FUNCTION_BLOCK FB_SlitPair_1
VAR_INPUT
    iBladeNegative: UINT; //Axis ID for negatively positioned blade
    iBladePositive: UINT; //Axis ID for positively positioned blade
    iGapSize: UINT; //Axis ID for the size of gap between slit blades
    iGapCentre: UINT; //Axis ID for the centre position of the gap formed by slit blades
    bEnable: BOOL; //Enable/disable the slit set
    bReset: BOOL; //Reset the slit set
    fEncoderScaling: LREAL := 10000; //default scaling denominator of 10000
    bAutoHome: BOOL := FALSE;
END_VAR
VAR_OUTPUT
    bEnabled: BOOL := FALSE; //Enabled status of function
    bError: BOOL; //Error status of function
    bHoming: BOOL := FALSE; //TRUE if function is homing axes
END_VAR
VAR
    eSlitPairState: E_SlitPairStates := E_SlitPairStates.INIT; //statemachine index

//Internal statuses for logic
    bResetting: BOOL := FALSE; //TRUE if axis going through a reset
    bRealAxesEnabled: BOOL := FALSE; //TRUE if all axes enabled
    bBladesHomed: BOOL:= FALSE; //TRUE if blade axes are calibrated
    bGapHomed: BOOL:= FALSE; //TRUE if virtual axes are calibrated
    bBladesCoupled: BOOL:= FALSE; //TRUE if both blade axes are coupled
    bBladesUncoupled: BOOL := FALSE; //TRUE if both blade axes are uncoupled
    bAxisErrorsPresent: BOOL := FALSE; //TRUE if error present on any real or virtual axis
    bFunctionInErrorState: BOOL := FALSE; //TRUE if function block is in one of the error related states
    fGapSizePosition: LREAL;
    iGapSizePosition AT %Q*: UDINT := 0;
    fGapCentrePosition: LREAL;
    iGapCentrePosition AT %Q*: UDINT := 0;
    resetCounterTimeout: UINT :=0;
    mcHomeGapSize: MC_Home;
    mcHomeGapCentre: MC_Home;
	fbSetPosGapsize: MC_SetPosition;
	fbSetPosGapCentre: MC_SetPosition;
	bSetPosiotnGap: BOOL := FALSE;
END_VAR

(* NOTES
For the virtual axis setup, the encoders need their type changed from "simulation encoder" to "Encoder (Universal)".
In addition the scale factor needs to be changed to a numerator of 1 and denominator of fEncoderScaling which is 10,000 by default)
Care needs to be taken with scaling and setup of both real and virtual axes to ensure velocities are not too fast and axes have time to settle before they submit a "complete move"
*)

//Configure homing routine of virtual axes
GVL.astAxes[iGapSize].stConfig.eHomeSeq := E_HomingRoutines.eHomeDirect;
GVL.astAxes[iGapCentre].stConfig.eHomeSeq := E_HomingRoutines.eHomeDirect;

//Run actions for slit set
actRunMethods(); //Update statuses
actErrorHandling(); //Error handling subroutine
actGapLimits(); //Set virtual axis limits to TRUE
actVirtualAxisPositions(); //Virtual axis encoder position subroutine


//Mc_Home FBs configured to clear homing signal
mcHomeGapSize(Axis := astAxes[iGapSize].Axis, HomingMode:=MC_HomingMode.MC_ResetCalibration);
mcHomeGapCentre(Axis:=astAxes[iGapCentre].Axis, HomingMode:=MC_HomingMode.MC_ResetCalibration);
mcHomeGapSize.Execute := FALSE;
mcHomeGapCentre.Execute := FALSE;

CASE eSlitPairState OF
    E_SlitPairStates.INIT:
        IF bEnable THEN
            eSlitPairState := E_SlitPairStates.INIT_CLEAR_GEARING;
        END_IF

    E_SlitPairStates.INIT_CLEAR_GEARING:
        actClearSlitGearing();
        eSlitPairState := E_SlitPairStates.INIT_GEAROUT_CHECK;

    E_SlitPairStates.INIT_GEAROUT_CHECK: //Check gearOut completion
        IF bBladesUncoupled THEN
            eSlitPairState := E_SlitPairStates.CHECK_HOME_STATUS;
        END_IF

    E_SlitPairStates.CHECK_HOME_STATUS: //If blades are already homed, skip to virtual homing, if blades not homed and autohome enabled then home blades, otherwise wait for blades to be homed
        IF bBladesHomed THEN
			eSlitPairState := E_SlitPairStates.HOME_GAP;
        ELSIF bRealAxesEnabled AND bAutoHome THEN
            eSlitPairState := E_SlitPairStates.HOME_BLADES; //If autohome enabled, home the blades
        END_IF

    E_SlitPairStates.HOME_BLADES: //Initiate homing of blade axes. Homing routine must be pre-configured by user
		mcHomeGapSize.Execute := TRUE;
        mcHomeGapCentre.Execute := TRUE;
        IF mcHomeGapSize.Done AND mcHomeGapCentre.Done THEN
       		GVL.astAxes[iBladeNegative].stControl.eCommand := E_MotionFunctions.eHome;
        	GVL.astAxes[iBladePositive].stControl.eCommand := E_MotionFunctions.eHome;
        	GVL.astAxes[iBladeNegative].stControl.bExecute := TRUE;
        	GVL.astAxes[iBladePositive].stControl.bExecute := TRUE;
        	bHoming := TRUE;
        	eSlitPairState := E_SlitPairStates.CHECK_BLADE_HOME_COMPLETE;    
        END_IF


    E_SlitPairStates.CHECK_BLADE_HOME_COMPLETE: //Wait for completion of blade homing routines
        IF bBladesHomed THEN
            eSlitPairState := E_SlitPairStates.HOME_GAP;
            bHoming := FALSE;
        END_IF

    E_SlitPairStates.HOME_GAP: //"Home" the virtual axes
        GVL.astAxes[iGapSize].stConfig.fHomePosition := fGapSizePosition;
        GVL.astAxes[iGapCentre].stConfig.fHomePosition := fGapCentrePosition;
        GVL.astAxes[iGapSize].stControl.eCommand := E_MotionFunctions.eHome;
        GVL.astAxes[iGapCentre].stControl.eCommand := E_MotionFunctions.eHome;
        GVL.astAxes[iGapSize].stControl.bExecute := TRUE;
        GVL.astAxes[iGapCentre].stControl.bExecute := TRUE;
        eSlitPairState := E_SlitPairStates.CHECK_GAP_HOME_COMPLETE;

    E_SlitPairStates.CHECK_GAP_HOME_COMPLETE: //Wait for virtual homing completion
        IF bGapHomed THEN
            eSlitPairState := E_SlitPairStates.GEARIN_SLITS;
        END_IF

    E_SlitPairStates.GEARIN_SLITS: //Setup gearing
        actSetupSlitGearing();
        eSlitPairState := E_SlitPairStates.CHECK_GEARIN_SLITS_COMPLETE;

    E_SlitPairStates.CHECK_GEARIN_SLITS_COMPLETE: //Wait for gearing complete
        IF bBladesCoupled THEN
            eSlitPairState := E_SlitPairStates.SLITS_OPERATIONAL;
        END_IF

    E_SlitPairStates.SLITS_OPERATIONAL: //SLITS OPERATIONAL - Monitor for any gear outs and re-gear when no busy blades
        bEnabled := TRUE;
		bSetPosiotnGap := FALSE;
        IF GVL.astAxes[iGapSize].stStatus.bBusy AND GVL.astAxes[iGapCentre].stStatus.bBusy THEN
			 eSlitPairState := E_SlitPairStates.SLITS_BUSY;
		END_IF

    E_SlitPairStates.SLITS_BUSY:
	 	IF GVL.astAxes[iGapSize].stStatus.bInTargetPosition AND GVL.astAxes[iGapCentre].stStatus.bInTargetPosition 
		   AND NOT GVL.astAxes[iBladePositive].stStatus.bMoving 
		   AND NOT GVL.astAxes[iBladeNegative].stStatus.bMoving THEN
			eSlitPairState := E_SlitPairStates.GEAROUT_BLADES;
		END_IF
		
	E_SlitPairStates.GEAROUT_BLADES: //Clear amy residual gearing
        actClearSlitGearing();
        eSlitPairState := E_SlitPairStates.CHECK_GEAROUT_COMPLETE;

    E_SlitPairStates.CHECK_GEAROUT_COMPLETE: //Check gearing cleared
        IF bBladesUncoupled THEN
            eSlitPairState := E_SlitPairStates.CLEAR_GAP_CALIBRATION; //MC_SetPosition, this ensures the setpoint position of the axis is updated.
        END_IF

    E_SlitPairStates.CLEAR_GAP_CALIBRATION:
        bSetPosiotnGap := TRUE; //this ensures the setpoint position of the axis is updated
        IF fbSetPosGapCentre.Done AND fbSetPosGapsize.Done THEN
			bSetPosiotnGap := FALSE;
            eSlitPairState := E_SlitPairStates.GEARIN_SLITS; //Back to gear_in
        END_IF

    E_SlitPairStates.ERROR: //ERROR STATE
		actClearSlitGearing();
		resetCounterTimeout := 0;
        bError := TRUE;
        bEnabled := FALSE;
        IF bReset THEN
            bResetting := TRUE;
            eSlitPairState := E_SlitPairStates.ERROR_GEAROUT;
        END_IF

    E_SlitPairStates.ERROR_GEAROUT: //Try to clear issues
        actClearSlitGearing();
        eSlitPairState := E_SlitPairStates.ERROR_GEAROUT_CHECK;

    E_SlitPairStates.ERROR_GEAROUT_CHECK:
        IF bBladesUncoupled THEN
            eSlitPairState := E_SlitPairStates.ERROR_RESET_AXES; 
        END_IF

    E_SlitPairStates.ERROR_RESET_AXES: //RESET ALL AXES
        GVL.astAxes[iBladeNegative].stControl.bReset := TRUE;
        GVL.astAxes[iBladePositive].stControl.bReset := TRUE;
        GVL.astAxes[iGapSize].stControl.bReset := TRUE;
        GVL.astAxes[iGapCentre].stControl.bReset := TRUE;
        resetCounterTimeout := resetCounterTimeout + 1;
        eSlitPairState := E_SlitPairStates.ERROR_RESET_CHECK;

    E_SlitPairStates.ERROR_RESET_CHECK:
	    GVL.astAxes[iBladeNegative].stControl.bReset := FALSE;
        GVL.astAxes[iBladePositive].stControl.bReset := FALSE;
        GVL.astAxes[iGapSize].stControl.bReset := FALSE;
        GVL.astAxes[iGapCentre].stControl.bReset := FALSE;
        IF resetCounterTimeout > 10 THEN
            eSlitPairState := E_SlitPairStates.ERROR;
            bResetting := FALSE;
            RETURN;
        END_IF
        IF bAxisErrorsPresent THEN
            eSlitPairState := E_SlitPairStates.ERROR_RESET_AXES;
        ELSE
            eSlitPairState := E_SlitPairStates.INIT;
            bError := FALSE;
            bResetting := FALSE;
        END_IF
END_CASE
bReset := FALSE;

fbSetPosGapCentre(
	Axis:= GVL.astAxes[iGapCentre].Axis, 
	Execute:= bSetPosiotnGap, 
	Position:= fGapCentrePosition, 
	Mode:= , 
	Options:= , 
	Done=> , 
	Busy=> , 
	Error=> , 
	ErrorID=> );
	
fbSetPosGapsize(
	Axis:= GVL.astAxes[iGapSize].Axis, 
	Execute:= bSetPosiotnGap, 
	Position:= fGapSizePosition, 
	Mode:= , 
	Options:= , 
	Done=> , 
	Busy=> , 
	Error=> , 
	ErrorID=> );

ACTION actClearSlitGearing:
//Action to send gearOut command to blade axes
GVL.astAxes[iBladeNegative].stControl.eCommand := E_MotionFunctions.eGearOut;
GVL.astAxes[iBladePositive].stControl.eCommand := E_MotionFunctions.eGearOut;
GVL.astAxes[iBladeNegative].stControl.bExecute := TRUE;
GVL.astAxes[iBladePositive].stControl.bExecute := TRUE;
END_ACTION

ACTION actErrorHandling:
//Error handling for slit functionality
IF bResetting THEN //ignore setting in error state if FB going through a reset
    RETURN;
END_IF

IF NOT bError AND bAxisErrorsPresent THEN
    eSlitPairState := E_SlitPairStates.ERROR;
END_IF
//IF eSlitPairState <> E_SlitPairStates.INIT AND NOT bRealAxesEnabled THEN
 //   eSlitPairState := E_SlitPairStates.ERROR;
//END_IF
IF (eSlitPairState <> E_SlitPairStates.INIT AND NOT bFunctionInErrorState) AND NOT bEnable THEN
    eSlitPairState := E_SlitPairStates.ERROR;
END_IF
//IF bEnabled AND NOT bBladesHomed THEN
//    eSlitPairState := E_SlitPairStates.ERROR;
//END_IF
END_ACTION

ACTION actGapLimits:
//Set Virtual axis inputs to TRUE to enable movement
GVL.astAxes[iGapSize].stInputs.bLimitFwd := GVL.astAxes[iBladePositive].stStatus.bFwEnabled AND GVL.astAxes[iBladeNegative].stStatus.bBwEnabled;
GVL.astAxes[iGapSize].stInputs.bLimitBwd := GVL.astAxes[iBladePositive].stStatus.bBwEnabled AND GVL.astAxes[iBladeNegative].stStatus.bFwEnabled;

GVL.astAxes[iGapCentre].stInputs.bLimitFwd := GVL.astAxes[iBladePositive].stStatus.bFwEnabled AND GVL.astAxes[iBladeNegative].stStatus.bFwEnabled;
GVL.astAxes[iGapCentre].stInputs.bLimitBwd := GVL.astAxes[iBladePositive].stStatus.bBwEnabled AND GVL.astAxes[iBladeNegative].stStatus.bBwEnabled;
END_ACTION

ACTION actRunMethods:
checkRealAxesEnabled(bOutput => bRealAxesEnabled);
checkBladesHomed(bOutput => bBladesHomed);
checkVirtualHomed(bOutput => bGapHomed);
checkBladesCoupled(bOutput => bBladesCoupled);
checkBladesUncoupled(bOutput => bBladesUncoupled);
checkAllAxisErrors(bOutput => bAxisErrorsPresent);
checkErrorState(bOutput => bFunctionInErrorState);
END_ACTION

ACTION actSetupSlitGearing:
GVL.astAxes[iBladeNegative].stControl.eCommand := E_MotionFunctions.eGearInMultiMaster;
GVL.astAxes[iBladeNegative].stConfig.astMultiMasterAxis[1].nIndex := iGapSize;
GVL.astAxes[iBladeNegative].stConfig.astMultiMasterAxis[1].fRatio := -0.5;
GVL.astAxes[iBladeNegative].stConfig.astMultiMasterAxis[2].nIndex := iGapCentre;
GVL.astAxes[iBladeNegative].stConfig.astMultiMasterAxis[2].fRatio := 1;
GVL.astAxes[iBladePositive].stControl.eCommand := E_MotionFunctions.eGearInMultiMaster;
GVL.astAxes[iBladePositive].stConfig.astMultiMasterAxis[1].nIndex := iGapSize;
GVL.astAxes[iBladePositive].stConfig.astMultiMasterAxis[1].fRatio := 0.5;
GVL.astAxes[iBladePositive].stConfig.astMultiMasterAxis[2].nIndex := iGapCentre;
GVL.astAxes[iBladePositive].stConfig.astMultiMasterAxis[2].fRatio := 1;
GVL.astAxes[iBladeNegative].stControl.bExecute := TRUE;
GVL.astAxes[iBladePositive].stControl.bExecute := TRUE;
END_ACTION

ACTION actVirtualAxisPositions:
(*Calculate virtual axis positions and convert to UDINT.
Conversion to UDINT is prohibited if it would exceed UDINT max value of 4,294,967,295.
If this is not done, it can cause overflow when connected to the encoder input and hard-crash the PLC which will only recover with a power cycle.
To preserve decimal position data of the LREAL (i.e. anything <1mm) it is necessary to scale the value before converting to UDINT.
This can be reversed with the correct scaling at the NC encoder level.
*)
fGapSizePosition := GVL.astAxes[iBladePositive].stStatus.fActPosition - GVL.astAxes[iBladeNegative].stStatus.fActPosition;
fGapCentrePosition := (GVL.astAxes[iBladePositive].stStatus.fActPosition + GVL.astAxes[iBladeNegative].stStatus.fActPosition) / 2;

IF bBladesHomed THEN
    IF ABS(fGapSizePosition) < 100000 THEN
        iGapSizePosition := LREAL_TO_UDINT(fGapSizePosition*fEncoderScaling);
    END_IF
    IF ABS(fGapCentrePosition) < 100000 THEN
        iGapCentrePosition := LREAL_TO_UDINT(fGapCentrePosition*fEncoderScaling);
    END_IF
END_IF
END_ACTION

(*Method to check if an error is present on any axis.
Returns TRUE if an error is present on any axis *)
METHOD checkAllAxisErrors: BOOL
VAR_OUTPUT
    bOutput: BOOL := FALSE;
END_VAR
IF GVL.astAxes[iGapSize].stStatus.bError THEN
    bOutput := TRUE;
END_IF
IF GVL.astAxes[iGapCentre].stStatus.bError THEN
    bOutput := TRUE;
END_IF
IF GVL.astAxes[iBladeNegative].stStatus.bError THEN
    bOutput := TRUE;
END_IF
IF GVL.astAxes[iBladePositive].stStatus.bError THEN
    bOutput := TRUE;
END_IF
END_METHOD

(*Method to check if both blades are coupled to the virtual axes.
Only returns TRUE if BOTH blades are coupled *)
METHOD checkBladesCoupled: BOOL
VAR_OUTPUT
    bOutput: BOOL := TRUE;
END_VAR
IF NOT GVL.astAxes[iBladeNegative].stStatus.bGeared THEN
    bOutput := FALSE;
END_IF
IF NOT GVL.astAxes[iBladePositive].stStatus.bGeared THEN
    bOutput := FALSE;
END_IF
END_METHOD

(*Method to check if blade axes are homed/have the calibration flag.
Only returns TRUE if BOTH blades are homed*)
METHOD checkBladesHomed: BOOL
VAR_OUTPUT
    bOutput: BOOL := TRUE;
END_VAR
IF NOT GVL.astAxes[iBladeNegative].stStatus.bHomed THEN
    bOutput := FALSE;
END_IF
IF NOT GVL.astAxes[iBladePositive].stStatus.bHomed THEN
    bOutput := FALSE;
END_IF
END_METHOD

(*Method to check if both blades are uncoupled from the virtual axes.
Only returns TRUE if BOTH blades are uncoupled *)
METHOD checkBladesUncoupled: BOOL
VAR_OUTPUT
    bOutput: BOOL:= TRUE;
END_VAR
IF GVL.astAxes[iBladeNegative].stStatus.bGeared THEN
    bOutput := FALSE;
END_IF
IF GVL.astAxes[iBladePositive].stStatus.bGeared THEN
    bOutput := FALSE;
END_IF
END_METHOD

METHOD checkErrorState: BOOL
VAR_OUTPUT
    bOutput: BOOL := FALSE;
END_VAR
IF eSlitPairState = E_SlitPairStates.ERROR THEN
    bOutput := TRUE;
END_IF
IF eSlitPairState = E_SlitPairStates.ERROR_GEAROUT THEN
    bOutput := TRUE;
END_IF
IF eSlitPairState = E_SlitPairStates.ERROR_GEAROUT_CHECK THEN
    bOutput := TRUE;
END_IF
IF eSlitPairState = E_SlitPairStates.ERROR_RESET_AXES THEN
    bOutput := TRUE;
END_IF
IF eSlitPairState = E_SlitPairStates.ERROR_RESET_CHECK THEN
    bOutput := TRUE;
END_IF
IF fbSetPosGapCentre.Error THEN
	bOutput := TRUE;
END_IF
IF fbSetPosGapSize.Error THEN
	bOutput := TRUE;
END_IF
END_METHOD

(*Method to check if all axes (real and virtual) are enabled.
Only returns TRUE if BOTH blades are homed*)
METHOD checkRealAxesEnabled: BOOL
VAR_OUTPUT
    bOutput: BOOL:= TRUE;
END_VAR
IF NOT GVL.astAxes[iBladeNegative].stStatus.bEnabled THEN
    bOutput := FALSE;
END_IF
IF NOT GVL.astAxes[iBladePositive].stStatus.bEnabled THEN
    bOutput := FALSE;
END_IF
END_METHOD

(*Method to check if the virtual axes for gap size and gap centre are homed/the calibration flag is present.
Only returns TRUE if BOTH virtual axes are homed *)
METHOD checkVirtualHomed: BOOL
VAR_OUTPUT
    bOutput: BOOL:= TRUE;
END_VAR
IF NOT GVL.astAxes[iGapSize].stStatus.bHomed THEN
    bOutput := FALSE;
END_IF
IF NOT GVL.astAxes[iGapCentre].stStatus.bHomed THEN
    bOutput := FALSE;
END_IF
END_METHOD

END_FUNCTION_BLOCK

(* stored: Version 1.1.0.1, ProductVersion 3.1.4024.11
   POU FB_SlitPair_1: Id {f51b9a67-df8e-44a7-b7a0-665c8fa1858b}, SpecialFunc None
   Action actClearSlitGearing: Id {3a4d22ec-7e5b-4e40-819d-256bca3488c2}
   Action actErrorHandling: Id {2e3499e1-91a1-4e6c-a0d9-62df7b2f6208}
   Action actGapLimits: Id {0e054f3c-c54c-49ec-8095-7757e8483915}
   Action actRunMethods: Id {a4d725de-6dce-4b2e-8f7f-739742e93dee}
   Action actSetupSlitGearing: Id {1be7f207-7970-4156-8ef0-fd25a353860f}
   Action actVirtualAxisPositions: Id {7a2cd7d0-03f7-4eb0-bed3-02cdb0852376}
   Method checkAllAxisErrors: Id {5075071e-fd77-4ab5-bbbe-0c78d8973eec}
   Method checkBladesCoupled: Id {e2dcbfdf-2f31-484f-8ca8-8b8014c4ffed}
   Method checkBladesHomed: Id {99df5367-edda-438a-8ea0-191775abd50f}
   Method checkBladesUncoupled: Id {2a27993f-38e3-44cb-83f7-f4b2169fcfa1}
   Method checkErrorState: Id {7c719146-4016-4f23-952a-a1b134152935}
   Method checkRealAxesEnabled: Id {ae693f74-a412-458c-b83c-2cd2bf8fc711}
   Method checkVirtualHomed: Id {b65d610d-f118-41e0-8166-59943c1ad868} *)
